FUNCTION_BLOCK L3_MachineAllocator (* Basic Function Block Type *)
  (* Standard: 61499-2 *)
  (* Version 0.0, 2014-11-06, EQUEROL, UJI *)
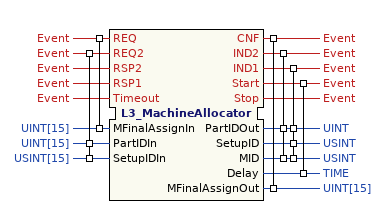
  EVENT_INPUT
    REQ WITH MFinalAssignIn; (* Normal Execution Request *)
    REQ2 WITH SetupIDIn, PartIDIn; (* Request from PPTable *)
    RSP2; (* Response from the PPTable *)
    RSP1; (* Response from the machine *)
    Timeout; (* Timeout expired *)
  END_EVENT
  EVENT_OUTPUT
    CNF WITH MFinalAssignOut; (* Request Confirm *)
    IND2 WITH PartIDOut, MID; (* Indicate to the PPTable that the setup was correctly assigned *)
    IND1 WITH MID, SetupID, PartIDOut; (* Send a setup to a machine *)
    Start WITH Delay; (* Timeout start *)
    Stop; (* Timeout stop *)
  END_EVENT
  VAR_INPUT
    MFinalAssignIn : ARRAY [0..14] OF UINT; (* Machine-PP Assignation vector *)
    PartIDIn : ARRAY [0..14] OF UINT; (* Part identifiers vector *)
    SetupIDIn : ARRAY [0..14] OF USINT; (* Setup identifiers vector *)
  END_VAR
  VAR_OUTPUT
    PartIDOut : UINT; (* Part identifier *)
    SetupID : USINT; (* Setup identifier *)
    MID : USINT; (* Machine identifier *)
    Delay : TIME; (* Timeout delay in ms *)
    MFinalAssignOut : ARRAY [0..14] OF UINT; (* Machine-PP Assignation vector *)
  END_VAR
  VAR
    AssignRemaining : BOOL := FALSE; (* Variable indicating if there is any setup to be assigned or not *)
    i : USINT; (* loop variable *)
    IFinalAssign : ARRAY [0..14] OF UINT := [0,0,0,0,0,0,0,0,0,0,0,0,0,0,0]; (* Internal Variable *)
    CurrentPartID : UINT := 0; (* Identifier of the part being assigned *)
    CurrentSetupID : USINT := 0; (* Identifier of the setup being assigned *)
    TOCounter : USINT := 0; (* Timeouts counter *)
  END_VAR
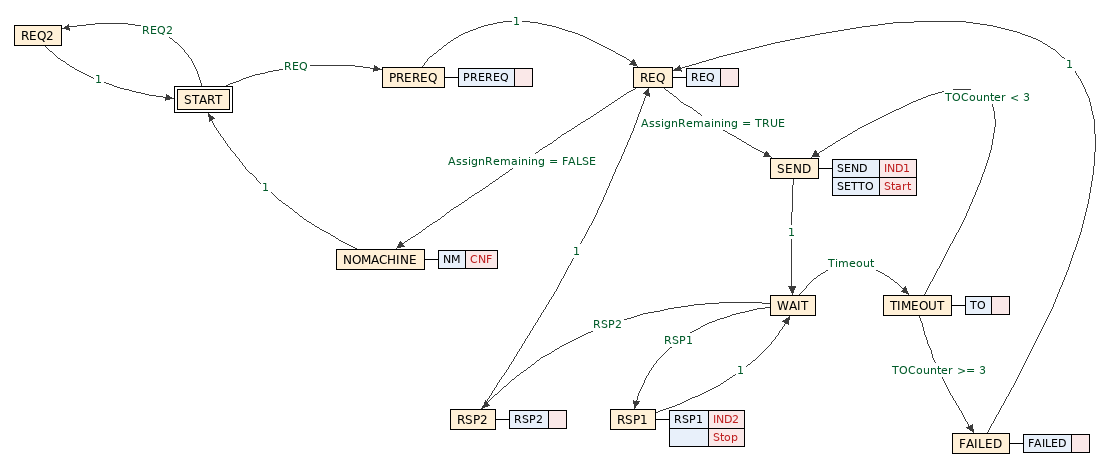
  EC_STATES
    START; (* Initial State *)
    REQ : REQ; (* Normal execution *)
    REQ2;
    SEND : SEND -> IND1, SETTO -> Start;
    PREREQ : PREREQ;
    NOMACHINE : NM -> CNF;
    WAIT;
    RSP1 : RSP1 -> IND2, -> Stop;
    TIMEOUT : TO;
    FAILED : FAILED;
    RSP2 : RSP2;
  END_STATES
  EC_TRANSITIONS
    START TO REQ2 := REQ2;
    REQ2 TO START := 1;
    START TO PREREQ := REQ;
    PREREQ TO REQ := 1;
    REQ TO NOMACHINE := AssignRemaining = FALSE;
    NOMACHINE TO START := 1;
    REQ TO SEND := AssignRemaining = TRUE;
    SEND TO WAIT := 1;
    RSP1 TO WAIT := 1;
    WAIT TO RSP1 := RSP1;
    WAIT TO TIMEOUT := Timeout;
    TIMEOUT TO SEND := TOCounter < 3;
    TIMEOUT TO FAILED := TOCounter >= 3;
    FAILED TO REQ := 1;
    WAIT TO RSP2 := RSP2;
    RSP2 TO REQ := 1;
  END_TRANSITIONS
  ALGORITHM REQ IN ST: (* Normally executed algorithm *)
AssignRemaining := FALSE;
WHILE ( i <15 AND NOT AssignRemaining ) DO
	(*Check if any part can be assigned to a machine*)
	IF (IFinalAssign[i] <> 0 ) AND (IFinalAssign[i] = PartIDIn[i]) THEN
		(*This part can be assigned*)
		CurrentPartID := PartIDIn[i];
		CurrentSetupID := SetupIDIn[i];
		AssignRemaining := TRUE;
	END_IF;
	i := i +1;
END_WHILE;
  END_ALGORITHM
  ALGORITHM SETTO IN ST: (* Timeout algorithm *)
Delay := TIME#1000ms;
  END_ALGORITHM
  ALGORITHM PREREQ IN ST: (* Algorithm to initialize internal variables for this request *)
FOR i:=0 TO 14 DO
	IFinalAssign[i] := MFinalAssignIn[i];
END_FOR;
i :=0;
  END_ALGORITHM
  ALGORITHM NM IN ST: (* No machine to be assigned algo *)
FOR i:=0 TO 14 DO
	 MFinalAssignOut[i] := IFinalAssign[i];
END_FOR;
  END_ALGORITHM
  ALGORITHM SEND IN ST: (* Assign setup algo *)
(*A setup needs to be assigned*)
PartIDOut:= CurrentPartID;
SetupID := CurrentSetupID;
(*MID is one based index, i is current machine +1*)
MID := i;
  END_ALGORITHM
  ALGORITHM RSP1 IN ST: (* Response from the machine algo *)
TOCounter := 0;
PartIDOut := CurrentPartID;
MID := i;
  END_ALGORITHM
  ALGORITHM TO IN ST: (* Timeout algo *)
TOCounter := TOCounter + 1;
  END_ALGORITHM
  ALGORITHM FAILED IN ST: (* FAILED algo *)
TOCounter := 0;
  END_ALGORITHM
  ALGORITHM RSP2 IN ST: (* Response from PPTable algo *)
(*Setup was succesfully assigned*)
IF i <> 0 THEN
	IFinalAssign[i-1] := 0;
END_IF;
  END_ALGORITHM
END_FUNCTION_BLOCK
